{attribute 'qualified_only'}
{attribute 'strict'}
TYPE E_RegulatorMode :
(
	eDisabled,
	ePID,
	eCascade
);
END_TYPE

(* stored: Version 1.1.0.1, ProductVersion 3.1.4024.12
   DUT E_RegulatorMode: Id {58f30ffc-65e3-46c2-a2e2-aea0c4b7c186} *)
